Staubli VAL3: refresh.pgx

program refresh()
// // page refresh
begin
    if  (nKey>=270 and nKey<=278) or use:bUseRefresh==true
    call refreshStatic()
    call buildList()
    call refreshDynamic()
    if abs(clock()-nRefresh)>nTime
      call refreshDynamic()
    endIf
  endIf
end
